FUNCTION_BLOCK FB_BINFILLER
VAR_INPUT
	UpLeftConveyor_IN		: ST_PD6_IN;
	UpRightConveyor_IN		: ST_PD6_IN;
	DownLeftConveyor_IN		: ST_PD6_IN;
	DownRightConveyor_IN	: ST_PD6_IN;
	Rotary_IN				: ST_PD6_IN;
	AugerLeft_IN			: ST_PD6_IN;
	AugerRight_IN			: ST_PD6_IN;
	Enable	: BOOL;
END_VAR
VAR_OUTPUT
	UpLeftConveyor		: FB_PD6;
	UpRightConveyor		: FB_PD6;
	DownLeftConveyor	: FB_PD6;
	DownRightConveyor	: FB_PD6;
	Rotary				: FB_PD6;
	AugerLeft			: FB_PD6;
	AugerRight			: FB_PD6;
END_VAR
VAR
	State		: (DEFAULT, INIT, IDLE, MANUAL, AUTO, ERROR);
	PrevState	: (DEFAULT, INIT, IDLE, MANUAL, AUTO, ERROR);
	StateEntry 	: BOOL;
END_VAR



IF State <> PrevState THEN
	StateEntry := TRUE;
	PrevState := State;
ELSE
	StateEntry := FALSE;
END_IF

CASE State OF
	DEFAULT:
		//
	INIT:
		//
	IDLE:
		//
	MANUAL:
		//
	AUTO:
		//
	ERROR:
		//
END_CASE

UpLeftConveyor(PD6_IN := UpLeftConveyor_IN);
UpRightConveyor(PD6_IN := UpRightConveyor_IN);
DownLeftConveyor(PD6_IN := DownLeftConveyor_IN);
DownRightConveyor(PD6_IN := DownRightConveyor_IN);
Rotary(PD6_IN := Rotary_IN);
AugerLeft(PD6_IN := AugerLeft_IN);
AugerRight(PD6_IN := AugerRight_IN);

END_FUNCTION_BLOCK

(* stored: Version 1.1.0.1, ProductVersion 3.1.4024.12
   POU FB_BINFILLER: Id {3099f396-b86b-4ba4-9528-44ca38af8d5b}, SpecialFunc None *)
